TYPE RtcSynchParams : 
STRUCT
    synchContextIdentity : ULINT;
    doSynch : BOOL;
    syncAmsId : STRING;
    syncPeriod : UINT;
END_STRUCT
END_TYPE

(* stored: Version 1.1.0.1
   DUT RtcSynchParams: Id {42dc72eb-0de2-035a-36d8-926288be288b} *)
